FUNCTION FUN_GetHighLowValue : UINT
VAR_INPUT
	nValue		:UINT;			// Actual value
END_VAR
VAR_OUTPUT
	nHigh		:UINT;			// True if value is greater than rLimitHigh
	nLow		:UINT;			// True if value is lower than rLimitLow	
END_VAR
VAR
END_VAR

IF nValue > nHigh THEN
	nHigh := nValue;
END_IF

IF nValue < nLow THEN
	nLow := nValue;
END_IF

END_FUNCTION

(* stored: Version 1.1.0.1, ProductVersion 3.1.4024.12
   POU FUN_GetHighLowValue: Id {524f67de-7bae-4d99-b66a-b211763d7c75}, SpecialFunc None *)
